(* PLC project new_comp, Dassault Systèmes ControlBuild 2024x Refresh1 *)
(* stored: creationDateTime 2024-04-10T10:54:19-01:00 *)

FUNCTION_BLOCK flask_motion_app.new_comp


ACTION C_source_code:

END_ACTION
END_FUNCTION_BLOCK
